(*********************************** G.D S.p.A. - Technical Department ***********************************
============= PROGRAM INFO ============
FOLDER:             TBD
MACHINES INVOLVED:  TBD 

============= DESCRIPTION =============
csp main interface program

============= REVISIONS ===============
Date		Version	 	Author      	Description             
----------	-------		------------  	--------------------------------------------
2019/09/27 	0000.00	 	M.Grasso		Creation of the PRG

**********************************************************************************************************)
PROGRAM _csp_case_glue_normal
VAR
END_VAR

(* CASE *)
	(* GLUE *)
		(* LS *)
		csp_case_glue_ls();
		(* OS *)
		csp_case_glue_os();
		(* SENSORS *)
		csp_case_glue_hotMelt_safety();

END_PROGRAM

(* stored: Version 1.1.0.1, ProductVersion 3.1.4024.3
   POU _csp_case_glue_normal: Id {651e871d-4514-4a71-b407-4a6cdb3db3e4}, SpecialFunc None *)
